(* CoDeSys 2.3 export: VEC3.EXP *)

(* Data type in MNG_TCPIP *)
TYPE VEC3 :(* 3d position *)
STRUCT
	x, y, z : REAL;
END_STRUCT
END_TYPE
